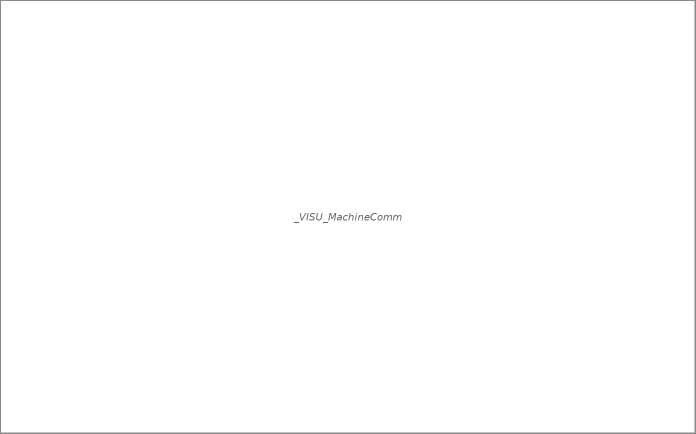
VISUALIZATION VISU_MACHINE  // 696x434
    Frame (0,0 696x434)
        shows _VISU_MachineComm(mInst := PRG_MACHINE.fbMachineComm)
END_VISUALIZATION

(* stored: Version 1.1.0.1, ProductVersion 3.1.4024.11
   Visu VISU_MACHINE: Id {3edaf7ab-1936-4338-b9d7-1d8cd9d9d5a8} *)
